{region '#Template'}
	{attribute 'Version' := '5.0.0.0'}
	{attribute 'Tags' := '"LCID": "1031", "Text": "Trade, Plant, General"'}
	{attribute 'Tags' := '"LCID": "1033", "Text": "Trade, Plant, General"'}
	{attribute 'Using' := '"Type": "Template", "URI": "Site"'}
	{attribute 'Description' := '"LCID": "1031", "Text": "Aufruf der Anlagen des Gewerks Allgemein"'}
	{attribute 'Description' := '"LCID": "1033", "Text": "Calling the plants of the trade general"'}
{endregion}
FUNCTION_BLOCK FB_BA_AutomationControl EXTENDS FB_BA_View
VAR_INPUT
END_VAR
VAR_INPUT CONSTANT
	Device				: FB_BA_Device;											 
	EvtGroups			: FB_BA_EvtGroupsAMEV2017;											 
	Cabinet				: FB_BA_ControlCabinet;				 
END_VAR

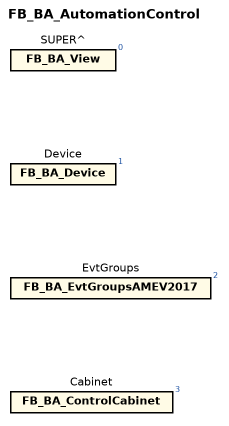
SUPER^(); // FB_BA_View
Device(); // FB_BA_Device
EvtGroups(); // FB_BA_EvtGroupsAMEV2017
Cabinet(); // FB_BA_ControlCabinet

METHOD FB_init : BOOL
VAR_INPUT
	bInitRetains : BOOL; // if TRUE, the retain variables are initialized (warm start / cold start)
	bInCopyCode : BOOL;  // if TRUE, the instance afterwards gets moved into the copy code (online change)
END_VAR
Device.iParent					:= THIS^;
Device.iLabel					:= LblPlt_Automation_control_equipment;	
Device.sObjectName				:= '{Idx=01}';  
Device.eDPADMode				:= E_BA_DPADMode.eInclude;		

EvtGroups.iParent				:= THIS^;	
EvtGroups.iLabel				:= LblPlt_EventGroups;
EvtGroups.sObjectName			:= '{Idx=01}';  
EvtGroups.eDPADMode				:= E_BA_DPADMode.eInclude;									

Cabinet.iParent					:= THIS^;	
Cabinet.iLabel					:= LblPlt_Control_cabinet;
Cabinet.sObjectName				:= '{Idx=01}';  
Cabinet.eDPADMode				:= E_BA_DPADMode.eInclude;
END_METHOD

END_FUNCTION_BLOCK

(* stored: Version 1.1.0.1, ProductVersion 3.1.4024.12
   POU FB_BA_AutomationControl: Id {3a11c574-07f3-4eac-bd2e-f348d461b6b2}, SpecialFunc None
   Method FB_init: Id {f7a1de78-1cc7-417a-8718-fb131f28a68a} *)
